FUNCTION_BLOCK Eventlogger
VAR
		Eventbuffer : ARRAY[0..MaxBuffersize] OF ST_Event;
		CurrentBufferIndex : INT :=0;
		_PersistentEventStorage : I_PersistentEventStorage;
END_VAR
VAR CONSTANT
	MaxBuffersize: INT := 100;
END_VAR

METHOD PUBLIC AddEvent : BOOL
VAR_INPUT
	eEventTypes: E_EventType;
	eEventSeverity: TcEventSeverity;
	eEventIdentity: UDINT;
	eEventText: STRING(255);
END_VAR
IF NOT IsEventBufferFull() THEN
	CurrentBufferIndex:=CurrentBufferIndex+1;
	Eventbuffer[CurrentBufferIndex].eEventTypes:=eEventTypes;
	Eventbuffer[CurrentBufferIndex].eEventSeverity:=eEventSeverity;
	Eventbuffer[CurrentBufferIndex].eEventIdentity:=eEventIdentity;
	Eventbuffer[CurrentBufferIndex].eEventText:=eEventText;
	UpdateEventTimeStamp(stEvent:=Eventbuffer[CurrentBufferIndex]);
	AddEvent:= TRUE;
ELSE
	AddEvent:= FALSE;
END_IF

//Store the event here
_PersistentEventStorage.StoreEvent(stEvent := Eventbuffer[CurrentBufferIndex]);
END_METHOD

METHOD FB_init : BOOL
VAR_INPUT
	bInitRetains : BOOL; // if TRUE, the retain variables are initialized (warm start / cold start)
	bInCopyCode : BOOL;  // if TRUE, the instance afterwards gets moved into the copy code (online change)
	iPersistentEventStorage:I_PersistentEventStorage;
END_VAR
_PersistentEventStorage:=iPersistentEventStorage;
END_METHOD

METHOD PRIVATE IsEventBufferFull : BOOL
IF (CurrentBufferIndex+1)> MaxBuffersize THEN
	IsEventBufferFull:=TRUE;
ELSE
	IsEventBufferFull:=FALSE;		
END_IF
END_METHOD

END_FUNCTION_BLOCK

(* stored: Version 1.1.0.1, ProductVersion 3.1.4024.12
   POU Eventlogger: Id {611a36b8-4b3d-43d9-b622-a5dca50e8044}, SpecialFunc None
   Method AddEvent: Id {d3d7941b-0ad0-4d03-b323-eac35cf7caeb}
   Method FB_init: Id {8eb6f229-87fc-4f89-ac3d-cf3349007c30}
   Method IsEventBufferFull: Id {01bc66bf-c64d-4e9b-bfdb-4c4d09f94f00} *)
